// TIA Portal V18 export
DATA_BLOCK "07_DOOR"   // DB8, F_DB
{ S7_Optimized_Access := 'TRUE'; DB_Accessible_From_OPC_UA := 'FALSE' }
VERSION : 0.1
// stored: AutoNumber true, DBAccessibleFromOPCUA false, DBAccessibleFromWebserver true
   VAR
      AlwaysFALSE : Bool;
      AlwaysTRUE : Bool;
      "No Operation" : Bool;
      "Door Closed SAFE_STATE [ =S1+SG1-B1 ]" : Bool;
      "Door Closed SAFE_STATE [ =S1+SG2-B1 ]" : Bool;
      "Door Closed SAFE_STATE [ =S2+SG3-B1 ]" : Bool;
      "Door Closed SAFE_STATE [ =S2+SG4-B1 ]" : Bool;
      "Door Closed DIAGNOSIS [ =S1+SG1-B1 ]" : Bool;
      "Door Closed DIAGNOSIS [ =S1+SG2-B1 ]" : Bool;
      "Door Closed DIAGNOSIS [ =S2+SG3-B1 ]" : Bool;
      "Door Closed DIAGNOSIS [ =S2+SG4-B1 ]" : Bool;
      "Door Alarm [ =S1+SG1-B1 ]" : Bool;
      "Door Alarm [ =S1+SG2-B1 ]" : Bool;
      "Door Alarm [ =S2+SG3-B1 ]" : Bool;
      "Door Alarm [ =S2+SG4-B1 ]" : Bool;
   END_VAR
BEGIN
END_DATA_BLOCK
